// TIA Portal V20 export
// export: Created 2025-12-01T14:57:28.8135412Z, ExportSetting None, DisplayName Totally Integrated Automation Portal, DisplayVersion V20 Update 3, DisplayName TIA Portal Openness, DisplayVersion V20 Update 3, DisplayName TIA Portal Version Control Interface, DisplayVersion V20 Update 3, DisplayName STEP 7 Professional, DisplayVersion V20 Update 3, DisplayName STEP 7 Safety, DisplayVersion V20 Update 2, DisplayName WinCC Basic/Comfort/Advanced, DisplayVersion V20 Update 3, DisplayName WinCC Professional, DisplayVersion V20 Update 3, DisplayName WinCC Unified, DisplayVersion V20 Update 3
FUNCTION "FC40_Llamadas_CB04" : Void   // FC40, LAD
{ S7_Optimized_Access := 'TRUE' }
// stored: AutoNumber false, SetENOAutomatically false
BEGIN

REGION Network 1: Control de Estado de Zona
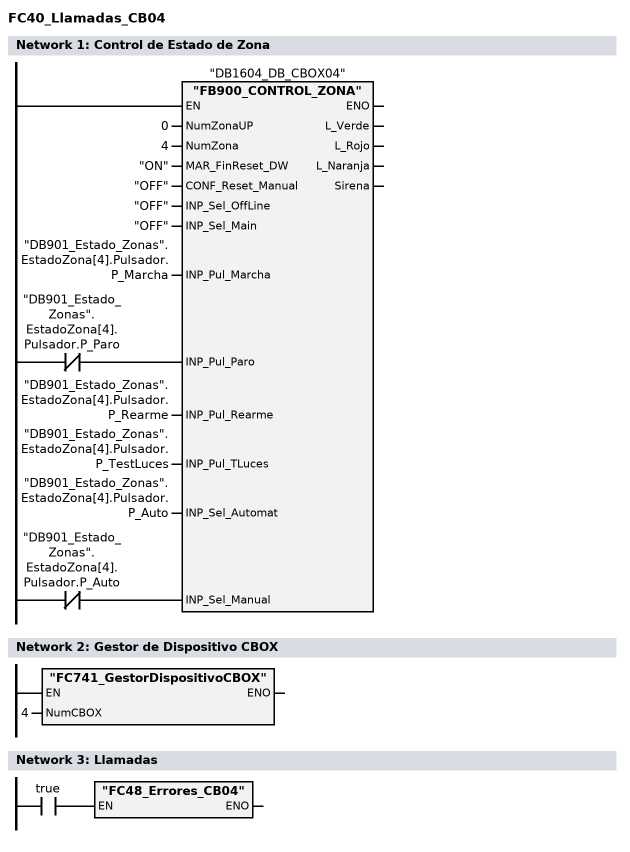
   RUNG wire#powerrail
      "DB1604_DB_CBOX04"(INP_Pul_Paro := wire#w1, INP_Sel_Manual := wire#w2, NumZonaUP := 0, NumZona := 4, MAR_FinReset_DW := "ON", CONF_Reset_Manual := "OFF", INP_Sel_OffLine := "OFF", INP_Sel_Main := "OFF", INP_Pul_Marcha := "DB901_Estado_Zonas".EstadoZona[4].Pulsador.P_Marcha, INP_Pul_Rearme := "DB901_Estado_Zonas".EstadoZona[4].Pulsador.P_Rearme, INP_Pul_TLuces := "DB901_Estado_Zonas".EstadoZona[4].Pulsador.P_TestLuces, INP_Sel_Automat := "DB901_Estado_Zonas".EstadoZona[4].Pulsador.P_Auto, L_Verde =>, L_Rojo =>, L_Naranja =>, Sirena =>)
   END_RUNG
   RUNG wire#powerrail
      I_Contact( "DB901_Estado_Zonas".EstadoZona[4].Pulsador.P_Paro )
   END_RUNG wire#w1
   RUNG wire#powerrail
      I_Contact( "DB901_Estado_Zonas".EstadoZona[4].Pulsador.P_Auto )
   END_RUNG wire#w2
   // the same network as SCL:
   "DB1604_DB_CBOX04"(NumZonaUP := 0,   // "FB900_CONTROL_ZONA"
                      NumZona := 4,
                      MAR_FinReset_DW := "ON",
                      CONF_Reset_Manual := "OFF",
                      INP_Sel_OffLine := "OFF",
                      INP_Sel_Main := "OFF",
                      INP_Pul_Marcha := "DB901_Estado_Zonas".EstadoZona[4].Pulsador.P_Marcha,
                      INP_Pul_Paro := NOT "DB901_Estado_Zonas".EstadoZona[4].Pulsador.P_Paro,
                      INP_Pul_Rearme := "DB901_Estado_Zonas".EstadoZona[4].Pulsador.P_Rearme,
                      INP_Pul_TLuces := "DB901_Estado_Zonas".EstadoZona[4].Pulsador.P_TestLuces,
                      INP_Sel_Automat := "DB901_Estado_Zonas".EstadoZona[4].Pulsador.P_Auto,
                      INP_Sel_Manual := NOT "DB901_Estado_Zonas".EstadoZona[4].Pulsador.P_Auto);
END_REGION

REGION Network 2: Gestor de Dispositivo CBOX
   RUNG wire#powerrail
      "FC741_GestorDispositivoCBOX"(NumCBOX := 4)
   END_RUNG
   // the same network as SCL:
   "FC741_GestorDispositivoCBOX"(NumCBOX := 4);
END_REGION

REGION Network 3: Llamadas
   RUNG wire#powerrail
      Contact( true )
      "FC48_Errores_CB04"()
   END_RUNG
   // the same network as SCL:
   IF true THEN "FC48_Errores_CB04"(); END_IF;
END_REGION
END_FUNCTION
